INTERFACE ITF_Component_HMI EXTENDS ITF_BaseComponent_HMI

METHOD LinkComponentData : BOOL
VAR_INPUT
	stData					: REFERENCE TO ST_Component_HMI_Link;
END_VAR
END_METHOD

END_INTERFACE

(* stored: Version 1.1.0.1, ProductVersion 3.1.4024.15
   Itf ITF_Component_HMI: Id {53d14405-dc04-4c14-986c-e6dfca1c6596}
   Method LinkComponentData: Id {e5e73123-96ac-4aa2-9edb-e5564f66e9d9} *)
